FUNCTION_BLOCK FB_ModbusSlave_Test EXTENDS FB_TestSuite
VAR
END_VAR

END_FUNCTION_BLOCK

(* stored: Version 1.1.0.1, ProductVersion 3.1.4024.12
   POU FB_ModbusSlave_Test: Id {a8a3ef86-486a-4869-be11-fdc0b5c73917}, SpecialFunc None *)
